(* IEC 61131-3 sources: AXOpen/src/core/ctrl/src/AxoRemoteTask, 1 file *)

(* ---- AxoRemoteTask.st ---- *)
NAMESPACE AXOpen.Core
    ///<summary>
    /// Provides a mechanism to exectute a logic from the PLC in an .NET environment.
    ///<remarks>
    ///> [!IMPORTANT]
    ///> The deferred execution in .NET envornment is not hard-real time nor deterministic.
    ///</remarks>
    ///</summary>
    {S7.extern=ReadWrite}
    CLASS PUBLIC AxoRemoteTask EXTENDS AxoTask
        VAR PUBLIC
            ///<summary>
            /// Remote system's done signature.
            /// When `StartSignature` and `DoneSignature` equal the task is considered executed on the remote system.
            ///</summary>
            DoneSignature : ULINT;

            ///<summary>
            /// Indicates whether this instance's remote procedure is initialized.
            ///</summary>
            ///<remarks>When the remote task is not initialized, but the execution is invoked, task enters error state.</remarks>
            IsInitialized : BOOL;

            HasRemoteException : BOOL;

            IsBeingCalledCounter : INT;

            {#ix-set:AttributeName = "<#RemoteTaskMessenger#>"}
            {#ix-set:PlcTextList =  "[1]:'<#Remote task is not initialized by remote partner.#>':'<#Make sure the remote application that should handle this remote request is running and is available to the controller.#>'';
                                    '[2]:'<#During the execution or remote task an error occured.#> |[[1]RemoteExceptionDetails]|':'<#Check detail of this remote task for more information about the problem.#>'"}
            _remoteTaskMessenger : AXOpen.Messaging.Static.AxoMessenger;

        END_VAR

        VAR PRIVATE
            _isInitialized : BOOL;
        END_VAR

        METHOD PUBLIC OVERRIDE Execute : BOOL
            VAR_INPUT
                inParent : IAxoObject;
            END_VAR

            Execute := SUPER.Execute(inParent);

            IF(NOT _isInitialized) THEN THIS._RemoteRestoreEnabled := TRUE; END_IF;
            _isInitialized := TRUE;

            _remoteTaskMessenger.Serve(THIS);

            IF(Execute) THEN
                _remoteTaskMessenger.ActivateOnCondition(UINT#1,NOT IsInitialized, AXOpen.Messaging.eAxoMessageCategory#Warning);
                //SUPER.ThrowWhen(NOT IsInitialized,'<#THE REMOTE TASK IS NOT INITIALIZED#>');
                SUPER.ThrowWhen(HasRemoteException, ErrorDetails);
                SUPER.DoneWhen(StartSignature = DoneSignature);
                // This will set the IsInitialized to TRUE when the remote system acknowledges the StartSignature
                // This will allow the task to be executed again in the future without going to error state
                IF(StartSignature = DoneSignature) THEN
                    THIS.IsInitialized := TRUE;
                END_IF;
                IsBeingCalledCounter := IsBeingCalledCounter + 1;
            END_IF;

            _remoteTaskMessenger.ActivateOnCondition(UINT#2,HasRemoteException, AXOpen.Messaging.eAxoMessageCategory#Error).RequireAcknowledgement();
        END_METHOD

        METHOD PUBLIC OVERRIDE Restore : IAxoTaskState
            SUPER.Restore();
            HasRemoteException := FALSE;
        END_METHOD

        // Internal use only!
        METHOD INTERNAL GetStartSignature : ULINT
            GetStartSignature := StartSignature;
        END_METHOD

        // Internal use only!
        METHOD INTERNAL SetDoneSignature
            DoneSignature := StartSignature;
        END_METHOD
    END_CLASS
END_NAMESPACE
